// TwinCAT 3 PLC project Parking_CO
// ProgramVersion: 3.1.4024.0
// libraries:
//   Tc2_Standard, * (Beckhoff Automation GmbH)
//   Tc2_System, * (Beckhoff Automation GmbH)
//   Tc3_Module, * (Beckhoff Automation GmbH)
//   VisuSymbols,3.5.10.0,System
// project tree:
//   / GlobalTextList.TcGTLO, PlcTask.TcTTO, Visualization Manager.TcVMO (not stored)
//   POUs/ MAIN.TcPOU
//   VISUs/ Visualization.TcVIS
// (motion and I/O tree: see PLC project trappenhuis_extraverlenging)
// real-time tasks:
//   TASK PlcTask: cycle T#10ms, priority 20, ADS port 350
//   TASK PlcTask1: cycle T#10ms, priority 21, ADS port 351
//   TASK PlcTask2: cycle T#10ms, priority 22, ADS port 352
//   TASK PlcTask3: cycle T#10ms, priority 23, ADS port 353
//   TASK PlcTask4: cycle T#10ms, priority 24, ADS port 354
//   TASK PlcTask5: cycle T#10ms, priority 25, ADS port 355
//   TASK PlcTask6: cycle T#10ms, priority 26, ADS port 356
//   TASK PlcTask7: cycle T#10ms, priority 27, ADS port 357
//   TASK PlcTask8: cycle T#10ms, priority 28, ADS port 358
//   TASK PlcTask9: cycle T#10ms, priority 29, ADS port 359
//   TASK PlcTask10: cycle T#10ms, priority 30, ADS port 360

CONFIGURATION Parking_CO
    RESOURCE PLC ON TwinCAT3
        TASK PlcTask(INTERVAL := T#10ms, PRIORITY := 30);
        PROGRAM MAIN WITH PlcTask : MAIN;
    END_RESOURCE
END_CONFIGURATION

// ---- POUs/MAIN.TcPOU
PROGRAM MAIN
VAR
	// Digitale ingangen
	bSensor1        AT %I*:BOOL;
	bSensor2        AT %I*:BOOL;
	Plus1auto       AT %I*:BOOL;
	Min1auto        AT %I*:BOOL;
	
	// Analoge ingangen 
	iAantalplaatsen AT %I*:WORD;
	
	// Digitale uitgangen
	bSlagboom       AT %Q*:BOOL;
	bGroen          AT %Q*:BOOL;
	bRood           AT %Q*:BOOL;
	
	// Analoge uitgangen 
	iTellerstand    AT %Q*:WORD;
	
	// Functies
	negatieveflankS2: F_TRIG;
	positieveflankS1: R_TRIG;
	positieveflankS2: R_TRIG;
	negatieveflankS1: F_TRIG;
	Aantalbezoekers : CTUD  ;
	
END_VAR

(*
Parking

Maak een visualisatie die de in- en uitgang van een parking voor personenwagens simuleert.

  - De toegang tot de parking wordt aangegeven door de verkeerslichten aan de ingang.
 	Als het maximum aantal parkeerplaatsen is bezet (zie tellerstand) moet het groene licht doven en het rode licht branden.
 
  - Bij het binnenrijden onderbreekt de wagen eerst sensor 1, 
	de slagboom opent en daarna wordt sensor 2 onderbroken. 
	Als de wagen verder naar binnenrijd wordt eerst sensor 1 terug vrijgegeven, 
	daarna wordt sensor 2 vrijgegeven. 
	Op dit moment wordt een wagen bij de tellerstand opgeteld en de slagboom wordt terug gesloten.
	
  - Bij het buiten rijden krijgen we de omgekeerde beweging. De wagen onderbreekt eerst sensor 2.
	De slagboom opent. Daarna wordt sensor 1 onderbroken. 
	Als de wagen naar buiten rijd wordt eerst sensor 2 terug vrijgegeven, daarna wordt sensor 1 vrijgegeven. 
	Op dit moment wordt een wagen van de tellerstand afgetrokken en de slagboom wordt terug gesloten.
*)

positieveflankS1(CLK:=bSensor1 , Q=> );
negatieveflankS1(CLK:=bSensor1 , Q=> );
positieveflankS2(CLK:=bSensor2 , Q=> );
negatieveflankS2(CLK:=bSensor2 , Q=> );
bSlagboom S=(positieveflankS1.Q AND NOT bSensor2)OR(positieveflankS2.Q AND NOT bSensor1);
bSlagboom R=(negatieveflankS2.Q AND NOT bSensor1)OR(negatieveflankS1.Q AND NOT bSensor2);

Aantalbezoekers(
	CU:=(positieveflankS1.Q AND NOT bSensor2)OR Plus1auto, 
	CD:=(positieveflankS2.Q AND NOT bSensor1)OR Min1auto , 
	RESET:= , 
	LOAD:= , 
	PV:= , 
	QU=> , 
	QD=> , 
	CV=>iTellerstand);
	
IF (iTellerstand >= iAantalplaatsen) THEN
	bRood:=TRUE;
	bGroen:=FALSE;
END_IF

IF (iTellerstand < iAantalplaatsen) THEN
	bGroen:=TRUE;
	bRood:=FALSE;
END_IF

END_PROGRAM

// ---- GlobalTextList.TcGTLO
TEXTLIST GlobalTextList
  53 = '%d'
  514 = '+1 auto'
  871 = '-1 auto'
  731 = 'Aantal bezoekers'
  759 = 'Aantal plaatsen'
END_TEXTLIST

// ---- VISUs/Visualization.TcVIS
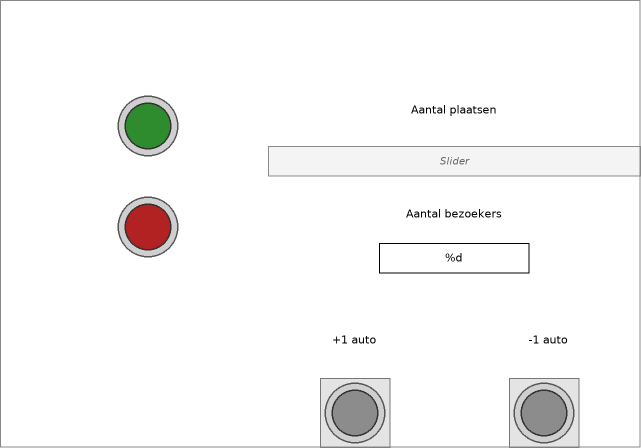
VISUALIZATION Visualization  // 641x448
    Slider (268,146 373x30), variable: MAIN.iAantalplaatsen, scale 0..100
    Rectangle (379,243 150x30), "%d", text variable: MAIN.iTellerstand, invisible if: MAIN.iTellerstand
        p4168582468: MAIN.iTellerstand
    Label (379,199 150x30), "Aantal bezoekers"
    Label (379,95 150x30), "Aantal plaatsen"
    Lamp1 (113,192 70x70), variable: MAIN.bRood, style: Lamp-Lamp1-Red
    Lamp1 (113,91 70x70), variable: MAIN.bGroen, style: Lamp-Lamp1-Green
    PushSwitch (320,378 70x70), variable: MAIN.Plus1auto, behaviour: TOGGLE, style: Switch-PushSwitch-Gray
    PushSwitch (509,378 70x70), variable: MAIN.Min1auto, behaviour: TOGGLE, style: Switch-PushSwitch-Gray
    Label (279,325 150x30), "+1 auto"
    Label (473,325 150x30), "-1 auto"
END_VISUALIZATION
